(* IEC 61131-3 sources: horner-cscape-mcp/artifacts/projects/ExportMCPProofProj/pous, 1 file *)

(* ---- ProofPOU.st ---- *)
PROGRAM ProofPOU
VAR
    nCount : INT := 0;
    bFlag : BOOL := TRUE;
END_VAR
nCount := nCount + 1;
END_PROGRAM
